{attribute 'GeneratedUsingTerminal: EL6692-0002-0016'}
{attribute addProperty BoxType "EL6692-0002-0016"}
{attribute addProperty Id "Sync_ModeAT %I*BYTE1TxPDO_toggleAT %I*BOOL1TxPDO_stateAT %I*BOOL1Control_value_update_toggleAT %I*BOOL1Timestamp_update_toggleAT %I*BOOL1External_device_not_connectedAT %I*BOOL1"}
{attribute addProperty CRC "1177473825"}
{attribute addProperty Size "6"}
TYPE SYNC_Inputs_462ED321 :
STRUCT
	{attribute addProperty Name "Sync_Mode"}
	Sync_Mode AT %I* : BYTE;
	{attribute addProperty Name "TxPDO_toggle"}
	TxPDO_toggle AT %I* : BOOL;
	{attribute addProperty Name "TxPDO_state"}
	TxPDO_state AT %I* : BOOL;
	{attribute addProperty Name "Control_value_update_toggle"}
	Control_value_update_toggle AT %I* : BOOL;
	{attribute addProperty Name "Timestamp_update_toggle"}
	Timestamp_update_toggle AT %I* : BOOL;
	{attribute addProperty Name "External_device_not_connected"}
	External_device_not_connected AT %I* : BOOL;
END_STRUCT
END_TYPE

(* stored: Version 1.2.0.0, ProductVersion 3.1.4024.9
   DUT SYNC_Inputs_462ED321: Id {21ccad92-0dd9-44aa-abd6-87dbf389ae13} *)
